(* Schneider Machine Expert - Basic project tank_level_ultrasonic_TM221CE16T, file version 3.0.0.0 *)
(* ProjectInformations: Name=Tank Level Control with Ultrasonic Sensor TM221CE16T with TM3AI4 *)

HARDWARE
  Cpu 0: TM221CE16T
  Extension 0: TM3AI4
  EthernetConfiguration: NetworkName=M221, IpAllocationMode=ByDhcp, IpAddress=192.168.1.10, SubnetMask=255.255.255.0
  SerialLineConfiguration: Baud=Baud19200, Parity=ParityEven, DataBits=DataBits8, StopBits=StopBits1, PhysicalMedium=PhysicalMediumRs485, TransmissionMode=TransmissionModeModbusRtu, SlaveId=1, Addressing=SlaveAddressing
  MastTask: UsePeriodScanMode=false, PeriodScan=100
  FastTask: Period=255
  CpuBehavior: StartingMode=StartAsPreviousState, AutoSaveRamOnEeprom=true, WatchdogPeriod=250

SYMBOLS  (address, symbol, comment, settings)
  %M0       PUMP_RUN  "Pump running latch with hysteresis"
  %M1       LEVEL_LOW  "Tank level below 1000mm from bottom"
  %M2       LEVEL_HIGH  "Tank level at 1500mm (500mm from sensor) - pump stop point"
  %MW0      LEVEL_RAW  "HMI Tag: Raw analog value from ultrasonic sensor (0-10000). Use for HMI: Read %IW1.0 directly via Modbus."
  %MW1      LEVEL_DISTANCE_MM  "HMI Tag: Distance from sensor in mm. Calculate in HMI: %IW1.0 / 2"
  %MW2      LEVEL_ACTUAL_MM  "HMI Tag: Actual level from tank bottom in mm. Calculate in HMI: 2000 - (%IW1.0 / 2)"
  %I0.0     PB_RESET  "Manual reset button"
  %I0.1     ESTOP  "Emergency stop (NC)"
  %Q0.0     PUMP_CONTACTOR  "Pump motor contactor"
  %Q0.1     LT_RUN  "Run indicator light"
  %Q0.2     LT_LOW_LEVEL  "Low level warning light"
  %IW1.0    ULTRASONIC_AIN  "Ultrasonic level transmitter 4-20mA. 5000mm range. Dead band 300mm. Raw 0-10000 = 0-5000mm distance."  [AIType=Current4_20mA, AIRange=Range0_10000, AIFilter=AIFilter4]

POU Tank Level Control
  (* SectionNumber=1 *)

// Rung 0: Low Level Detection
// Ultrasonic sensor: 5000mm range = 10000 raw. Distance = Raw/2. Level from bottom = 2000mm - Distance. Raw greater than 2000 means distance greater than 1000mm, so level less than 1000mm from bottom.
  LD [%IW1.0>2000]        (* ULTRASONIC_AIN *)
  ST %M1                  (* LEVEL_LOW *)
  // as ST:
  //   LEVEL_LOW := ULTRASONIC_AIN>2000;
  (* the ladder stored for this rung does not match its IL; not drawn *)

// Rung 1: High Level Detection
// Pump stop point: 500mm from transmitter. Raw = 500 x 2 = 1000. When raw less than 1000, level is 1500mm from bottom (500mm from sensor). Stop pumping.
  LD [%IW1.0<1000]        (* ULTRASONIC_AIN *)
  ST %M2                  (* LEVEL_HIGH *)
  // as ST:
  //   LEVEL_HIGH := ULTRASONIC_AIN<1000;
  (* the ladder stored for this rung does not match its IL; not drawn *)

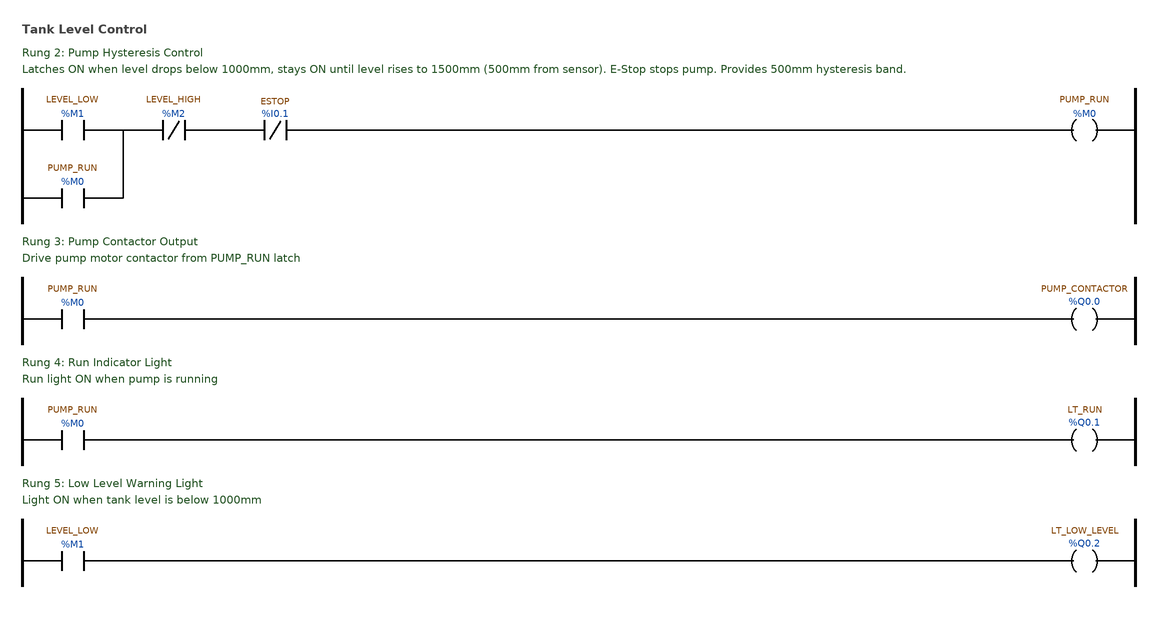

// Rung 2: Pump Hysteresis Control
// Latches ON when level drops below 1000mm, stays ON until level rises to 1500mm (500mm from sensor). E-Stop stops pump. Provides 500mm hysteresis band.
  LD %M1                  (* LEVEL_LOW *)
  OR %M0                  (* PUMP_RUN *)
  ANDN %M2                (* LEVEL_HIGH *)
  ANDN %I0.1              (* ESTOP *)
  ST %M0                  (* PUMP_RUN *)
  // as ST:
  //   PUMP_RUN := (LEVEL_LOW OR PUMP_RUN) AND NOT LEVEL_HIGH AND NOT ESTOP;

// Rung 3: Pump Contactor Output
// Drive pump motor contactor from PUMP_RUN latch
  LD %M0                  (* PUMP_RUN *)
  ST %Q0.0                (* PUMP_CONTACTOR *)
  // as ST:
  //   PUMP_CONTACTOR := PUMP_RUN;

// Rung 4: Run Indicator Light
// Run light ON when pump is running
  LD %M0                  (* PUMP_RUN *)
  ST %Q0.1                (* LT_RUN *)
  // as ST:
  //   LT_RUN := PUMP_RUN;

// Rung 5: Low Level Warning Light
// Light ON when tank level is below 1000mm
  LD %M1                  (* LEVEL_LOW *)
  ST %Q0.2                (* LT_LOW_LEVEL *)
  // as ST:
  //   LT_LOW_LEVEL := LEVEL_LOW;
